// Examples of objects that refer different event classes.
// > One object per 'EventType' and 'AlarmMode'.
// > One "PlantLock" per 'EventType'.
// > One "PlantLock" for entire view.
// > See "FB_BA_EC01" to view decleared event classes.
// [Hint]
// > All reference-variables are implemented to ease monitoring of relevant variables.
FUNCTION_BLOCK FB_Evt_Events EXTENDS FB_BA_View
VAR
	{region 'General'}
		Lock					: FB_BA_PlantLock				:= (iParent:=THIS^);
	{endregion}
		 
	{region 'Alarm'}
		Alm						: FB_BA_View					:= (iParent:=THIS^,	sDescription:= '[Alarm]');
			AlmLock				: FB_BA_PlantLock				:= (iParent:=Alm);
							
			BIAlmSmpl_Val		: REFERENCE TO BOOL				REF= BIAlmSmpl.bVal;
			BIAlmSmpl_LockPrio	: POINTER TO E_BA_LockPriority	:= ADR(BIAlmSmpl.eEnPlantLock);
			BIAlmSmpl			: FB_BA_BI						:= (iParent:=Alm,	iLabel:=MyLabels.Cmd,	iProfile:=MyProfiles.CmdB,	nEventClassID:=12);
			BIAlmStd_Val		: REFERENCE TO BOOL				REF= BIAlmStd.bVal;
			BIAlmStd_LockPrio	: POINTER TO E_BA_LockPriority	:= ADR(BIAlmStd.eEnPlantLock);
			BIAlmStd			: FB_BA_BI						:= (iParent:=Alm,	iLabel:=MyLabels.Cmd,	iProfile:=MyProfiles.CmdB,	nEventClassID:=11,	eEnPlantLock:= E_BA_LockPriority.eHigh);
			BIAlmExt_Val		: REFERENCE TO BOOL				REF= BIAlmExt.bVal;
			BIAlmExt_LockPrio	: POINTER TO E_BA_LockPriority	:= ADR(BIAlmExt.eEnPlantLock);
			BIAlmExt			: FB_BA_BI						:= (iParent:=Alm,	iLabel:=MyLabels.Cmd,	iProfile:=MyProfiles.CmdB,	nEventClassID:=10);
	{endregion}
	{region 'Disturb'}
		Dstb					: FB_BA_View					:= (iParent:=THIS^,	sDescription:= '[Disturb]');
			DstbLock			: FB_BA_PlantLock				:= (iParent:=Dstb);

			BIDstbSmpl_Val		: REFERENCE TO BOOL				REF= BIDstbSmpl.bVal;
			BIDstbSmpl_LockPrio	: POINTER TO E_BA_LockPriority	:= ADR(BIDstbSmpl.eEnPlantLock);
			BIDstbSmpl			: FB_BA_BI						:= (iParent:=Dstb,	iLabel:=MyLabels.Cmd,	iProfile:=MyProfiles.CmdB,	nEventClassID:=52);
			BIDstbStd_Val		: REFERENCE TO BOOL				REF= BIDstbStd.bVal;
			BIDstbStd_LockPrio	: POINTER TO E_BA_LockPriority	:= ADR(BIDstbStd.eEnPlantLock);
			BIDstbStd			: FB_BA_BI						:= (iParent:=Dstb,	iLabel:=MyLabels.Cmd,	iProfile:=MyProfiles.CmdB,	nEventClassID:=51,	eEnPlantLock:= E_BA_LockPriority.eMedium);
			BIDstbExt_Val		: REFERENCE TO BOOL				REF= BIDstbExt.bVal;
			BIDstbExt_LockPrio	: POINTER TO E_BA_LockPriority	:= ADR(BIDstbExt.eEnPlantLock);
			BIDstbExt			: FB_BA_BI						:= (iParent:=Dstb,	iLabel:=MyLabels.Cmd,	iProfile:=MyProfiles.CmdB,	nEventClassID:=50);
	{endregion}
	{region 'Maintenance'}
		Mntn					: FB_BA_View					:= (iParent:=THIS^,	sDescription:= '[Maintenance]');
			MntnLock			: FB_BA_PlantLock				:= (iParent:=Mntn);

			BIMntnSmpl_Val		: REFERENCE TO BOOL				REF= BIMntnSmpl.bVal;
			BIMntnSmpl_LockPrio	: POINTER TO E_BA_LockPriority	:= ADR(BIMntnSmpl.eEnPlantLock);
			BIMntnSmpl			: FB_BA_BI						:= (iParent:=Mntn,	iLabel:=MyLabels.Cmd,	iProfile:=MyProfiles.CmdB,	nEventClassID:=92);
			BIMntnStd_Val		: REFERENCE TO BOOL				REF= BIMntnStd.bVal;
			BIMntnStd_LockPrio	: POINTER TO E_BA_LockPriority	:= ADR(BIMntnStd.eEnPlantLock);
			BIMntnStd			: FB_BA_BI						:= (iParent:=Mntn,	iLabel:=MyLabels.Cmd,	iProfile:=MyProfiles.CmdB,	nEventClassID:=91,	eEnPlantLock:= E_BA_LockPriority.eLocalHigh);
			BIMntnExt_Val		: REFERENCE TO BOOL				REF= BIMntnExt.bVal;
			BIMntnExt_LockPrio	: POINTER TO E_BA_LockPriority	:= ADR(BIMntnExt.eEnPlantLock);
			BIMntnExt			: FB_BA_BI						:= (iParent:=Mntn,	iLabel:=MyLabels.Cmd,	iProfile:=MyProfiles.CmdB,	nEventClassID:=90);
	{endregion}
	{region 'Notification'}
		Ntfy					: FB_BA_View					:= (iParent:=THIS^,	sDescription:= '[Notification]');
			NtfyLock			: FB_BA_PlantLock				:= (iParent:=Ntfy);

			BINtfySmpl_Val		: REFERENCE TO BOOL				REF= BINtfySmpl.bVal;
			BINtfySmpl_LockPrio	: POINTER TO E_BA_LockPriority	:= ADR(BINtfySmpl.eEnPlantLock);
			BINtfySmpl			: FB_BA_BI						:= (iParent:=Ntfy,	iLabel:=MyLabels.Cmd,	iProfile:=MyProfiles.CmdB,	nEventClassID:=132);
			BINtfyStd_Val		: REFERENCE TO BOOL				REF= BINtfyStd.bVal;
			BINtfyStd_LockPrio	: POINTER TO E_BA_LockPriority	:= ADR(BINtfyStd.eEnPlantLock);
			BINtfyStd			: FB_BA_BI						:= (iParent:=Ntfy,	iLabel:=MyLabels.Cmd,	iProfile:=MyProfiles.CmdB,	nEventClassID:=131,	eEnPlantLock:= E_BA_LockPriority.eLocalMedium);
	{endregion}
	{region 'Other'}
		Other					: FB_BA_View					:= (iParent:=THIS^,	sDescription:= '[Other]');
			OtherLock			: FB_BA_PlantLock				:= (iParent:=Other);
				 
			BIOthrSmpl_Val		: REFERENCE TO BOOL				REF= BIOthrSmpl.bVal;
			BIOthrSmpl_LockPrio	: POINTER TO E_BA_LockPriority	:= ADR(BIOthrSmpl.eEnPlantLock);
			BIOthrSmpl			: FB_BA_BI						:= (iParent:=Other,	iLabel:=MyLabels.Cmd,	iProfile:=MyProfiles.CmdB,	nEventClassID:=182);
			BIOthrStd_Val		: REFERENCE TO BOOL				REF= BIOthrStd.bVal;
			BIOthrStd_LockPrio	: POINTER TO E_BA_LockPriority	:= ADR(BIOthrStd.eEnPlantLock);
			BIOthrStd			: FB_BA_BI						:= (iParent:=Other,	iLabel:=MyLabels.Cmd,	iProfile:=MyProfiles.CmdB,	nEventClassID:=181);
	{endregion}                                                
END_VAR

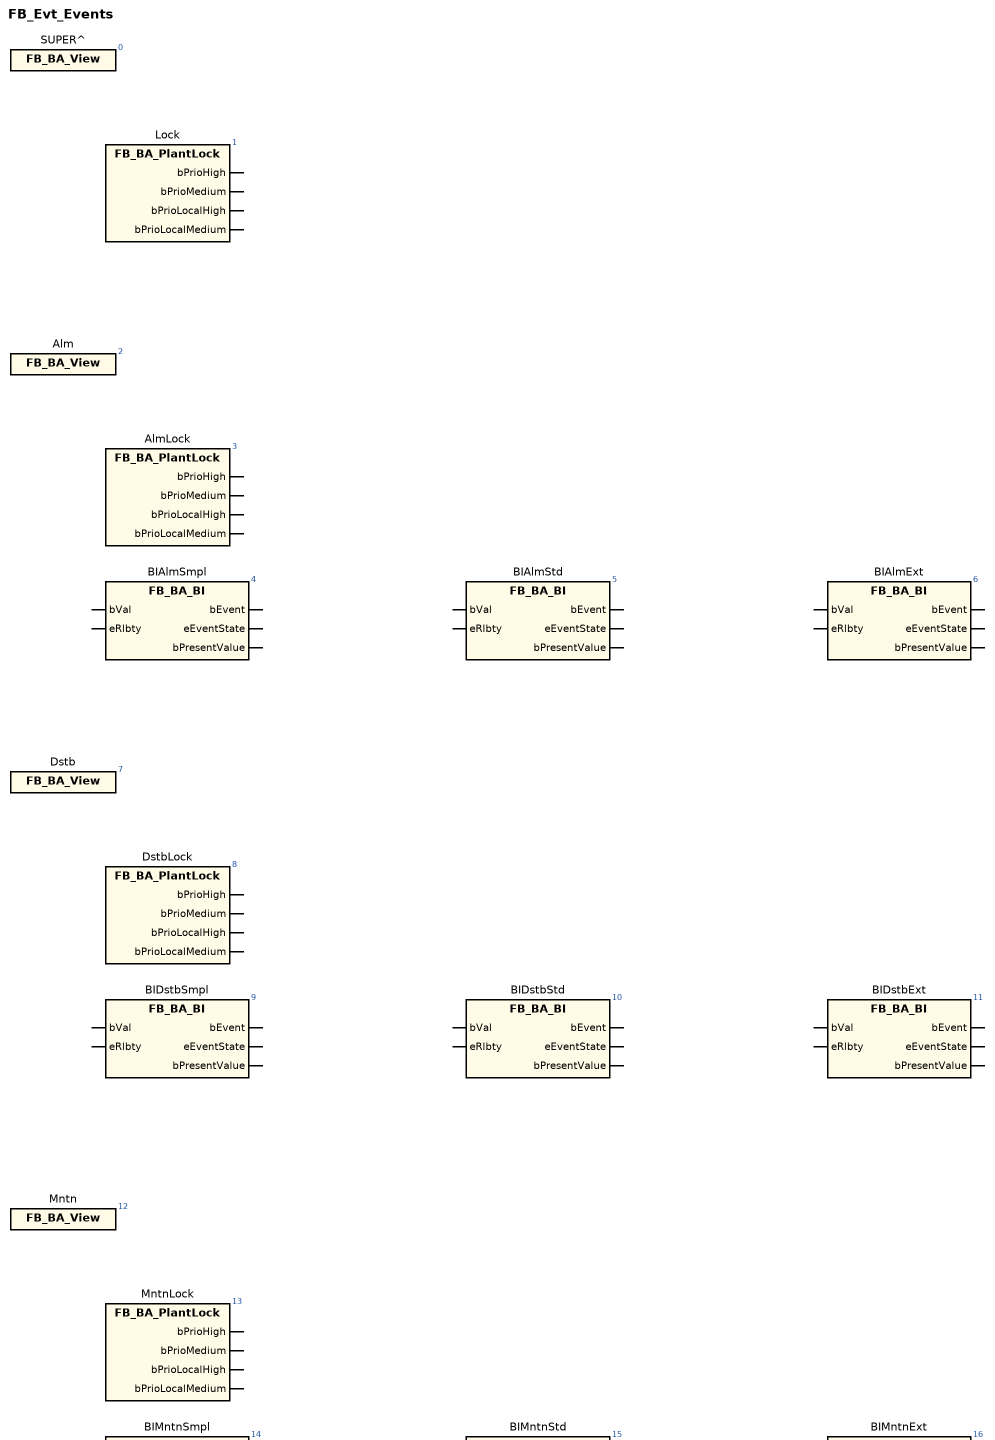
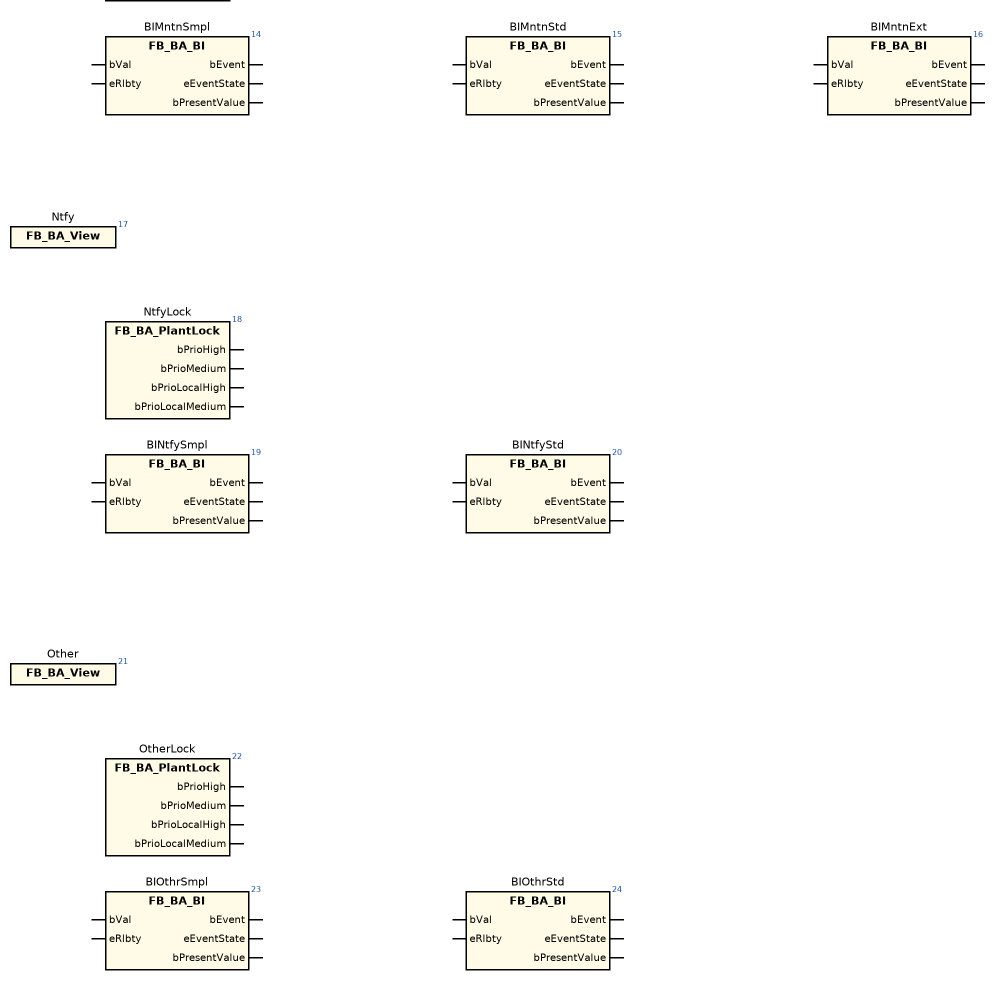
SUPER^(); // FB_BA_View
Lock(); // FB_BA_PlantLock
Alm(); // FB_BA_View
AlmLock(); // FB_BA_PlantLock
BIAlmSmpl(); // FB_BA_BI
BIAlmStd(); // FB_BA_BI
BIAlmExt(); // FB_BA_BI
Dstb(); // FB_BA_View
DstbLock(); // FB_BA_PlantLock
BIDstbSmpl(); // FB_BA_BI
BIDstbStd(); // FB_BA_BI
BIDstbExt(); // FB_BA_BI
Mntn(); // FB_BA_View
MntnLock(); // FB_BA_PlantLock
BIMntnSmpl(); // FB_BA_BI
BIMntnStd(); // FB_BA_BI
BIMntnExt(); // FB_BA_BI
Ntfy(); // FB_BA_View
NtfyLock(); // FB_BA_PlantLock
BINtfySmpl(); // FB_BA_BI
BINtfyStd(); // FB_BA_BI
Other(); // FB_BA_View
OtherLock(); // FB_BA_PlantLock
BIOthrSmpl(); // FB_BA_BI
BIOthrStd(); // FB_BA_BI

END_FUNCTION_BLOCK

(* stored: Version 1.1.0.1, ProductVersion 3.1.4024.5
   POU FB_Evt_Events: Id {b218198f-fd5a-469c-b5b5-684d23708b65}, SpecialFunc None *)
